FUNCTION alg_a_HledQ1 : BOOL
VAR_INPUT
	state: STATE;
END_VAR

alg_a_HledQ1 := FALSE;

END_FUNCTION

(* stored: Version 1.1.0.1, ProductVersion 3.1.4022.18
   POU alg_a_HledQ1: Id {eef45d93-3288-4fd6-819f-bcda7e35e49c}, SpecialFunc None *)
